PROGRAM Dosificador_Polvo_2
VAR
	fbDosificador_P2 :Equipo_Motor_ATV320;
	Balanza_P2_WT1: Balanza;
	fbTR_P2_VI: Equipo_Motor_ATV320;
	TararP2:BOOL;
	dHS:DINT;
	
	Tmr_Alr_ZeroSpeed: TON;
	TDemoraInyectarPolvo: TON;
	Tiempo_seg_to_TIME_TDemoraInyec: Tiempo_seg_to_TIME;
	Auxtdemora: TIME;
	Calc_Veloc_Polvo_2: Calc_Veloc_Polvo;
	Tiempo_seg_to_TIME_TInyeccion: Tiempo_seg_to_TIME;
	AuxInyec: TIME;
	TInyeccion: TON;
	ModoCalibrarP2 :BOOL;
	
	InyectarCalibrarP2: BOOL;
	Calibracion_Po_calc_P2: Calibracion_Po_calc;
	PolvoAsociado:STRING;
	TR_P2_WT1_rValue_REAL: REAL;
	TON_SolicitaPo: TON;
END_VAR
VAR PERSISTENT
	UltimaCalibracao	:UDINT;	//Data da ultima calibração feita com sucesso
END_VAR
VAR // added by the converter: edge detectors and wires of the graphical bodies
    _w1, _w2, _w3 : BOOL;
    _ft1 : F_TRIG;
    _rt1 : R_TRIG;
END_VAR

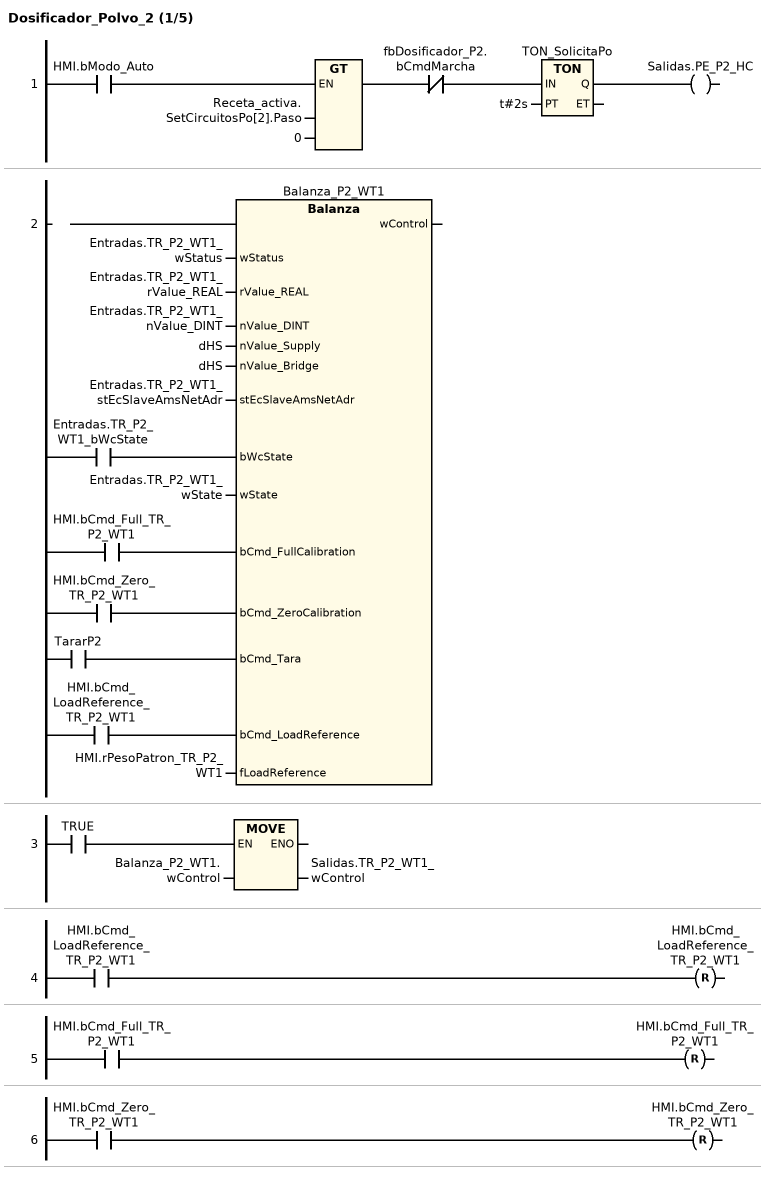
// NETWORK 1
TON_SolicitaPo(IN := (HMI.bModo_Auto AND Receta_activa.SetCircuitosPo[2].Paso > 0) AND NOT fbDosificador_P2.bCmdMarcha, PT := t#2s); // TON
Salidas.PE_P2_HC := TON_SolicitaPo.Q;

// NETWORK 2
Balanza_P2_WT1(
    wStatus := Entradas.TR_P2_WT1_wStatus,
    rValue_REAL := Entradas.TR_P2_WT1_rValue_REAL,
    nValue_DINT := Entradas.TR_P2_WT1_nValue_DINT,
    nValue_Supply := dHS,
    nValue_Bridge := dHS,
    stEcSlaveAmsNetAdr := Entradas.TR_P2_WT1_stEcSlaveAmsNetAdr,
    bWcState := Entradas.TR_P2_WT1_bWcState,
    wState := Entradas.TR_P2_WT1_wState,
    bCmd_FullCalibration := HMI.bCmd_Full_TR_P2_WT1,
    bCmd_ZeroCalibration := HMI.bCmd_Zero_TR_P2_WT1,
    bCmd_Tara := TararP2,
    bCmd_LoadReference := HMI.bCmd_LoadReference_TR_P2_WT1,
    fLoadReference := HMI.rPesoPatron_TR_P2_WT1); // Balanza

// NETWORK 3
Salidas.TR_P2_WT1_wControl := Balanza_P2_WT1.wControl;

// NETWORK 4
HMI.bCmd_LoadReference_TR_P2_WT1 R= HMI.bCmd_LoadReference_TR_P2_WT1;

// NETWORK 5
HMI.bCmd_Full_TR_P2_WT1 R= HMI.bCmd_Full_TR_P2_WT1;

// NETWORK 6
HMI.bCmd_Zero_TR_P2_WT1 R= HMI.bCmd_Zero_TR_P2_WT1;

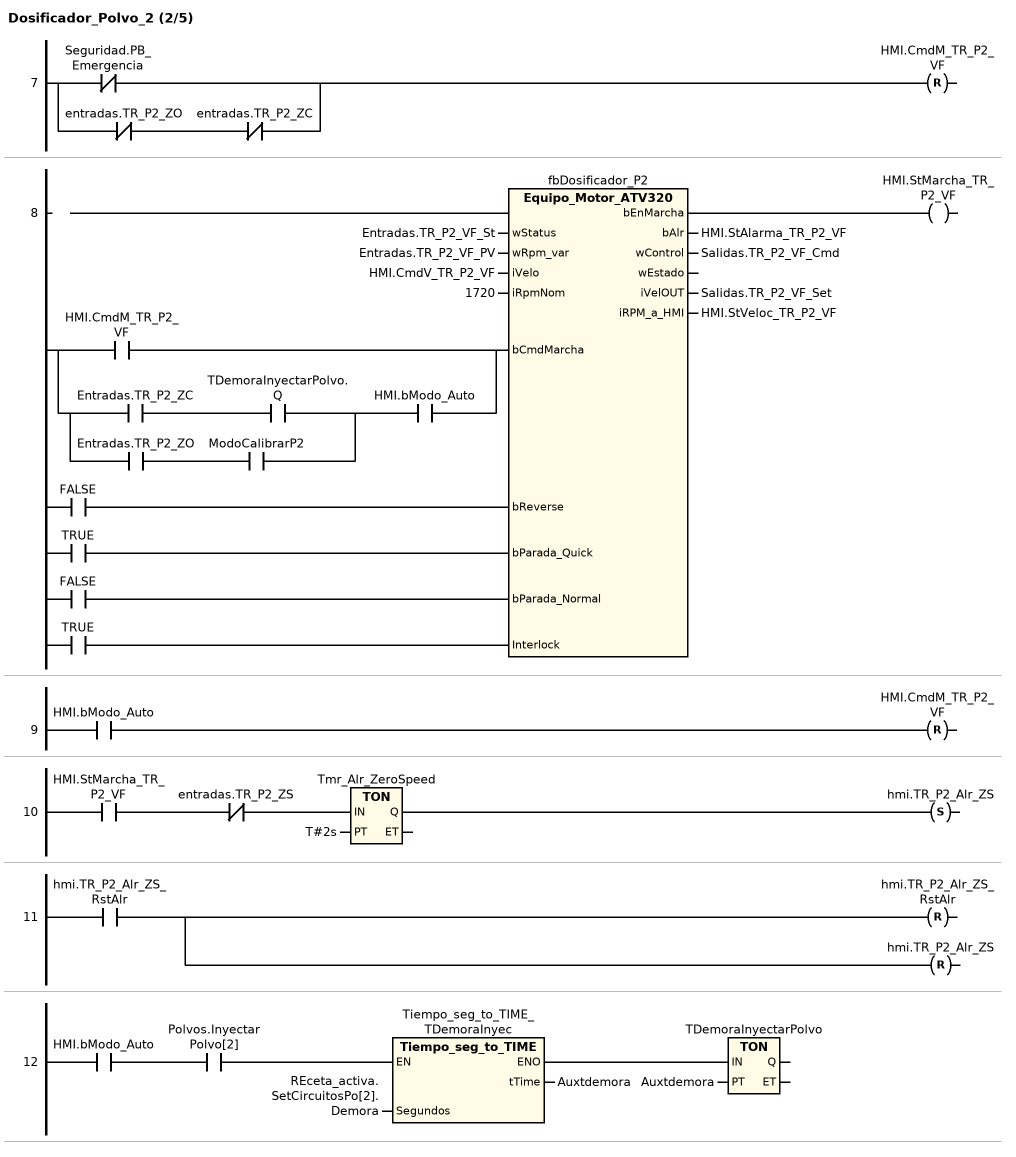
// NETWORK 7
HMI.CmdM_TR_P2_VF R= NOT Seguridad.PB_Emergencia OR NOT entradas.TR_P2_ZO AND NOT entradas.TR_P2_ZC;

// NETWORK 8
fbDosificador_P2(
    wStatus := Entradas.TR_P2_VF_St,
    wRpm_var := Entradas.TR_P2_VF_PV,
    iVelo := HMI.CmdV_TR_P2_VF,
    iRpmNom := 1720,
    bCmdMarcha := HMI.CmdM_TR_P2_VF OR (Entradas.TR_P2_ZC AND TDemoraInyectarPolvo.Q OR Entradas.TR_P2_ZO AND ModoCalibrarP2) AND HMI.bModo_Auto,
    bReverse := FALSE,
    bParada_Quick := TRUE,
    bParada_Normal := FALSE,
    Interlock := TRUE,
    bAlr => HMI.StAlarma_TR_P2_VF,
    wControl => Salidas.TR_P2_VF_Cmd,
    iVelOUT => Salidas.TR_P2_VF_Set,
    iRPM_a_HMI => HMI.StVeloc_TR_P2_VF); // Equipo_Motor_ATV320
HMI.StMarcha_TR_P2_VF := fbDosificador_P2.bEnMarcha;

// NETWORK 9
HMI.CmdM_TR_P2_VF R= HMI.bModo_Auto;

// NETWORK 10
Tmr_Alr_ZeroSpeed(IN := HMI.StMarcha_TR_P2_VF AND NOT entradas.TR_P2_ZS, PT := T#2s); // TON
hmi.TR_P2_Alr_ZS S= Tmr_Alr_ZeroSpeed.Q;

// NETWORK 11
_w1 := hmi.TR_P2_Alr_ZS_RstAlr;
hmi.TR_P2_Alr_ZS_RstAlr R= _w1;
hmi.TR_P2_Alr_ZS R= _w1;

// NETWORK 12
_w2 := HMI.bModo_Auto AND Polvos.InyectarPolvo[2];
IF _w2 THEN
    Tiempo_seg_to_TIME_TDemoraInyec(Segundos := REceta_activa.SetCircuitosPo[2].Demora, tTime => Auxtdemora); // Tiempo_seg_to_TIME
END_IF
TDemoraInyectarPolvo(IN := _w2, PT := Auxtdemora); // TON

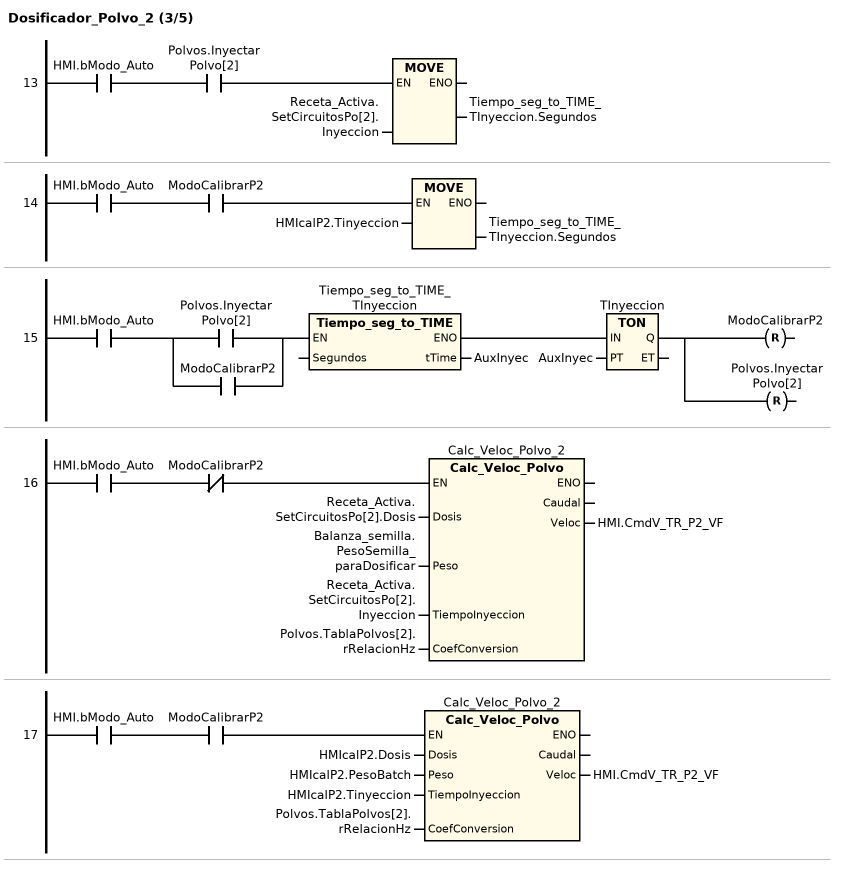
// NETWORK 13
IF HMI.bModo_Auto AND Polvos.InyectarPolvo[2] THEN
    Tiempo_seg_to_TIME_TInyeccion.Segundos := Receta_Activa.SetCircuitosPo[2].Inyeccion;
END_IF

// NETWORK 14
IF HMI.bModo_Auto AND ModoCalibrarP2 THEN Tiempo_seg_to_TIME_TInyeccion.Segundos := HMIcalP2.Tinyeccion; END_IF

// NETWORK 15
_w3 := HMI.bModo_Auto AND (Polvos.InyectarPolvo[2] OR ModoCalibrarP2);
IF _w3 THEN
    Tiempo_seg_to_TIME_TInyeccion(tTime => AuxInyec); // Tiempo_seg_to_TIME
END_IF
TInyeccion(IN := _w3, PT := AuxInyec); // TON
ModoCalibrarP2 R= TInyeccion.Q;
Polvos.InyectarPolvo[2] R= TInyeccion.Q;

// NETWORK 16
IF HMI.bModo_Auto AND NOT ModoCalibrarP2 THEN
    Calc_Veloc_Polvo_2(
        Dosis := Receta_Activa.SetCircuitosPo[2].Dosis,
        Peso := Balanza_semilla.PesoSemilla_paraDosificar,
        TiempoInyeccion := Receta_Activa.SetCircuitosPo[2].Inyeccion,
        CoefConversion := Polvos.TablaPolvos[2].rRelacionHz,
        Veloc => HMI.CmdV_TR_P2_VF); // Calc_Veloc_Polvo
END_IF

// NETWORK 17
IF HMI.bModo_Auto AND ModoCalibrarP2 THEN
    Calc_Veloc_Polvo_2(
        Dosis := HMIcalP2.Dosis,
        Peso := HMIcalP2.PesoBatch,
        TiempoInyeccion := HMIcalP2.Tinyeccion,
        CoefConversion := Polvos.TablaPolvos[2].rRelacionHz,
        Veloc => HMI.CmdV_TR_P2_VF); // Calc_Veloc_Polvo
END_IF

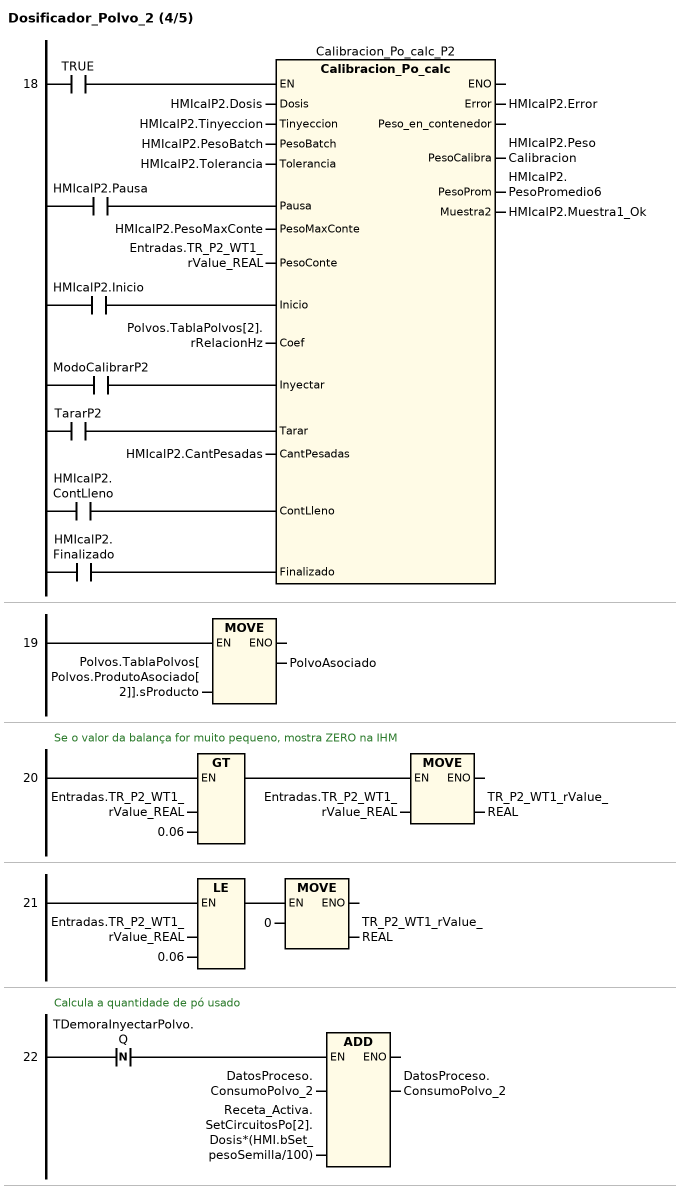
// NETWORK 18
Calibracion_Po_calc_P2(
    Dosis := HMIcalP2.Dosis,
    Tinyeccion := HMIcalP2.Tinyeccion,
    PesoBatch := HMIcalP2.PesoBatch,
    Tolerancia := HMIcalP2.Tolerancia,
    Pausa := HMIcalP2.Pausa,
    PesoMaxConte := HMIcalP2.PesoMaxConte,
    PesoConte := Entradas.TR_P2_WT1_rValue_REAL,
    Inicio := HMIcalP2.Inicio,
    Coef := Polvos.TablaPolvos[2].rRelacionHz,
    Inyectar := ModoCalibrarP2,
    Tarar := TararP2,
    CantPesadas := HMIcalP2.CantPesadas,
    ContLleno := HMIcalP2.ContLleno,
    Finalizado := HMIcalP2.Finalizado,
    Error => HMIcalP2.Error,
    PesoCalibra => HMIcalP2.PesoCalibracion,
    PesoProm => HMIcalP2.PesoPromedio6,
    Muestra2 => HMIcalP2.Muestra1_Ok); // Calibracion_Po_calc

// NETWORK 19
PolvoAsociado := Polvos.TablaPolvos[Polvos.ProdutoAsociado[2]].sProducto;

// NETWORK 20
// Se o valor da balança for muito pequeno, mostra ZERO na IHM
IF Entradas.TR_P2_WT1_rValue_REAL > 0.06 THEN TR_P2_WT1_rValue_REAL := Entradas.TR_P2_WT1_rValue_REAL; END_IF

// NETWORK 21
IF Entradas.TR_P2_WT1_rValue_REAL <= 0.06 THEN TR_P2_WT1_rValue_REAL := 0; END_IF

// NETWORK 22
// Calcula a quantidade de pó usado
_ft1(CLK := TDemoraInyectarPolvo.Q);
IF _ft1.Q THEN
    DatosProceso.ConsumoPolvo_2 := DatosProceso.ConsumoPolvo_2 + (Receta_Activa.SetCircuitosPo[2].Dosis*(HMI.bSet_pesoSemilla/100));
END_IF

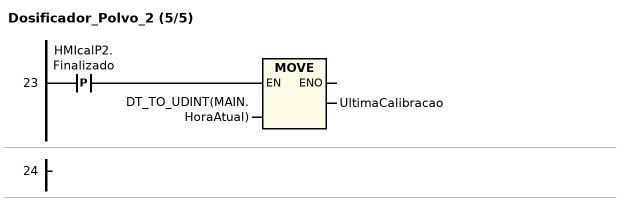
// NETWORK 23
_rt1(CLK := HMIcalP2.Finalizado);
IF _rt1.Q THEN UltimaCalibracao := DT_TO_UDINT(MAIN.HoraAtual); END_IF

// NETWORK 24

END_PROGRAM

(* stored: Version 1.1.0.1, ProductVersion 3.1.4024.14
   POU Dosificador_Polvo_2: Id {b0b84098-eec7-4727-a54e-0cd50b333d46}, SpecialFunc None *)
